// TIA Portal V18 export
DATA_BLOCK "Function Ratio check"   // DB43
{ S7_Optimized_Access := 'TRUE' }
VERSION : 0.1
// stored: AutoNumber false, DBAccessibleFromOPCUA true, IsOnlyStoredInLoadMemory false, IsRetainMemResEnabled false, IsWriteProtectedInAS false, MemoryReserve 100
   VAR RETAIN
      input : Struct
         "Set Flowrate" : Real := 15.0;
         "Set time" : DInt := 0;
         "Flowrate adjustment A" : Real := 0.0;
         "Flowrate adjustment B" : Real := 0.0;
         "set qty" : Real := 1.0;
         Mode : Int := 0;
      END_STRUCT;
   END_VAR
   VAR
      Control : Struct
         "Start metering" : Bool := FALSE;
         "Stop metering" : Bool := FALSE;
         "metering running" : Bool := FALSE;
         "metering completed" : Bool := FALSE;
         "start refill" : Bool := FALSE;
         "quick stop" : Bool := FALSE;
         ProgressBar_Limit : DInt := 4000;
         ProgressBar : DInt := 0;
         AcceptValue : Bool := FALSE;
         ShowPopup : Bool := FALSE;
      END_STRUCT;
      output : Struct
         "ON_pump A" : Bool := FALSE;
         "ON_pump B" : Bool := FALSE;
         ON_mixer : Bool := FALSE;
         "ON_outlet Valve A" : Bool := FALSE;
         "Running time" : Int := 0;
         "ON_outlet valve B" : Bool := FALSE;
         "Volume dispensed" : Real := 0.0;
         "ON_inlet A" : Bool := FALSE;
         "ON_inlet B" : Bool := FALSE;
         "Flowrate running" : Real := 0.0;
         "Remaing qty to dispense" : Real := 0.0;
      END_STRUCT;
   END_VAR
   VAR RETAIN
      PumpCaliberationControls : Struct
         CurrentSet_A : Real := 0.0;
         CurrentSet_B : Real := 0.0;
         CurrentActual_A : Real := 0.0;
         CurrentActual_B : Real := 0.0;
         "CurrentActual_A Gram" : Real := 0.0;
         "CurrentActual_B Gram" : Real := 0.0;
         CurrentSetFlowrate_A : Real := 0.0;
         CurrentSetFlowrate_B : Real := 0.0;
      END_STRUCT;
      PumpCaliberationPara : Struct
         CurrentDeviation_A : Real := 0.0;
         CurrrentDeviation_B : Real := 0.0;
         TotalDeviation_A : Real := 0.0;
         TotalDeviation_B : Real := 0.0;
         "Delete Calibration_A" : Bool := FALSE;
         "Delete Calibration_B" : Bool := FALSE;
      END_STRUCT;
   END_VAR
   VAR
      Parametes : Struct
         AddedMixingRatio : Real := 0.0;
      END_STRUCT;
   END_VAR
BEGIN
END_DATA_BLOCK
